// TwinCAT 3 PLC project PLC
// ProgramVersion: 3.1.4023.0
// libraries:
//   Tc3_Module, * (Beckhoff Automation GmbH)
// project tree:
//   DUTs/ Celsius.TcDUT, Fahrenheit.TcDUT, mbar.TcDUT, mmHg.TcDUT, Pascal.TcDUT, PoundsPerSquareInch.TcDUT, TerminalStatus.TcDUT, Torr.TcDUT
//   / MAIN.TcPOU, PlcTask.TcTTO
//   POUs/ FahrenheitToCelsius.TcPOU, IsValid.TcPOU, mmHgToPascal.TcPOU, PoundsPerSquareInchToPascal.TcPOU, TorrToMbar.TcPOU, TorrToMbarWithAlias.TcPOU, TorrToMbarWithUnits.TcPOU
// real-time tasks:
//   TASK PlcTask: cycle T#10ms, priority 20, ADS port 350

CONFIGURATION PLC
    RESOURCE PLC ON TwinCAT3
        TASK PlcTask(INTERVAL := T#10ms, PRIORITY := 20);
        PROGRAM MAIN WITH PlcTask : MAIN;
    END_RESOURCE
END_CONFIGURATION

// ---- DUTs/Celsius.TcDUT
TYPE Celsius EXTENDS TerminalStatus :
STRUCT
    _ : REAL;
END_STRUCT
END_TYPE

// ---- DUTs/Fahrenheit.TcDUT
TYPE Fahrenheit EXTENDS TerminalStatus :
STRUCT
    _ : LREAL; 
END_STRUCT
END_TYPE

// ---- DUTs/mbar.TcDUT
TYPE mbar : REAL; END_TYPE

// ---- DUTs/mmHg.TcDUT
TYPE mmHg :
STRUCT
    _ : REAL;
    unit : STRING := 'mmHg';
END_STRUCT
END_TYPE

// ---- DUTs/Pascal.TcDUT
TYPE Pascal :
STRUCT
    _ : REAL;
END_STRUCT
END_TYPE

// ---- DUTs/PoundsPerSquareInch.TcDUT
TYPE PoundsPerSquareInch :
STRUCT
     _ : REAL;
END_STRUCT
END_TYPE

// ---- DUTs/TerminalStatus.TcDUT
TYPE TerminalStatus :
STRUCT
    WorkingCounterError : BOOL;
    IOError : BOOL;
END_STRUCT
END_TYPE

// ---- DUTs/Torr.TcDUT
TYPE Torr : REAL; END_TYPE

// ---- MAIN.TcPOU
PROGRAM MAIN
VAR
    maximumPressure : REAL; // [mbar]
	
    pressure1 : REAL; // [mbar]
	pressure2 : REAL; // [Torr]
    
    pressure1_mbar : REAL;
    pressure2_Torr : REAL;
    
    pressure_si : mbar;
    pressure_imperial : Torr;
    
    pressure_eu : Pascal;
    pressure_us : PoundsPerSquareInch;
    
    pressure_hg : mmHg := (_:=0.31456);
    pressure_pa : Pascal; 
    
    temperature_eu : Celsius;
    temperature_us : Fahrenheit := (_:=104);
    
    temperature_eu_error : Celsius;
    temperature_us_error : Fahrenheit := (_:=97, IOError:=TRUE);
END_VAR

maximumPressure := 1E5;
pressure2 := TorrToMbar(pressure:=pressure1);
pressure2_Torr := TorrToMbarWithUnits(pressure_Torr:=pressure1_mbar);
pressure_imperial := TorrToMbarWithAlias(pressure:=pressure_si);
//// This raises a compiler warning 
//pressure_us := PoundsPerSquareInchToPascal(pressure:=pressure_eu);
pressure_pa := mmHgToPascal(pressure:=pressure_hg);
temperature_eu := FahrenheitToCelsius(temperature_us);
temperature_eu_error := FahrenheitToCelsius(temperature_us_error);

END_PROGRAM

// ---- POUs/TorrToMbar.TcPOU
FUNCTION TorrToMbar : REAL
VAR_INPUT
    pressure : REAL; // Torr
END_VAR

TorrToMbar := pressure * 1.3332236842;

END_FUNCTION

// ---- POUs/TorrToMbarWithUnits.TcPOU
FUNCTION TorrToMbarWithUnits : REAL
VAR_INPUT
    pressure_Torr : REAL;
END_VAR

TorrToMbarWithUnits := pressure_Torr * 1.3332236842;

END_FUNCTION

// ---- POUs/TorrToMbarWithAlias.TcPOU
FUNCTION TorrToMbarWithAlias : mbar
VAR_INPUT
    pressure : Torr;
END_VAR

TorrToMbarWithAlias := pressure * 1.3332236842;

END_FUNCTION

// ---- POUs/mmHgToPascal.TcPOU
FUNCTION mmHgToPascal : Pascal
VAR_INPUT
     pressure : mmHg;
END_VAR

mmHgToPascal._ := pressure._ * 133322;

END_FUNCTION

// ---- POUs/FahrenheitToCelsius.TcPOU
FUNCTION FahrenheitToCelsius : Celsius
VAR_INPUT
    temperature : Fahrenheit;
END_VAR

FahrenheitToCelsius.IOError := temperature.IOError;
FahrenheitToCelsius.WorkingCounterError := temperature.WorkingCounterError;
IF IsValid(temperature) THEN
    FahrenheitToCelsius._ := (temperature._ - 32) /  1.8;
END_IF

END_FUNCTION

// ---- POUs/IsValid.TcPOU
FUNCTION IsValid : BOOL
VAR_INPUT
    status : TerminalStatus;
END_VAR

IsValid := NOT (status.IOError OR status.WorkingCounterError);

END_FUNCTION

// ---- POUs/PoundsPerSquareInchToPascal.TcPOU
FUNCTION PoundsPerSquareInchToPascal : Pascal
VAR_INPUT
    pressure : PoundsPerSquareInch;
END_VAR

PoundsPerSquareInchToPascal._ := pressure._ * 6895;

END_FUNCTION
